(* IEC 61131-3 sources: simple-control-modules/src/Bulbs, 3 files *)

(* ---- Colors.st ---- *)
NAMESPACE Simatic.Ax.SimpleControlModules
    TYPE
        Colors : (Red, Green, Blue, Yellow);
    END_TYPE

END_NAMESPACE

(* ---- Bulb.st ---- *)
USING Simatic.Ax.Io.Output;
USING Simatic.Ax.Io.Input;

NAMESPACE Simatic.Ax.SimpleControlModules

    /// Class to handle a bulb
    CLASS Bulb
        VAR PUBLIC
            Output : ItfBinOutput;
        END_VAR

        /// Switch the lamp on (value := TRUE) or off (value := FALSE)
        /// value : Value to set
        METHOD PUBLIC Set
            VAR_INPUT
                value : bool;
            END_VAR
            IF (Output = NULL) THEN
                RETURN;
            END_IF;
            Output.SetQ(value := value);

        END_METHOD

        /// Switch the lamp on
        METHOD PUBLIC SwitchOn
            IF (Output = NULL) THEN
                RETURN;
            END_IF;
            Output.SetQ(value := TRUE);
        END_METHOD

        /// Switch the lamp off
        METHOD PUBLIC SwitchOff
            IF (Output = NULL) THEN
                RETURN;
            END_IF;
            Output.SetQ(value := FALSE);
        END_METHOD

        /// Toggle the lamp
        METHOD PUBLIC Toggle
            IF (Output = NULL) THEN
                RETURN;
            END_IF;
            Output.Toggle();
        END_METHOD

    END_CLASS
END_NAMESPACE

(* ---- LightStack.st ---- *)
USING Simatic.Ax.IO.Output;

NAMESPACE Simatic.Ax.SimpleControlModules

    /// Class of a lightstack with 3 lamps (Red, Yellow, Green)

    CLASS LightStackRdYeGnBl
        VAR PUBLIC
            QRed : ItfBinOutput;
            QYellow : ItfBinOutput;
            QGreen : ItfBinOutput;
            QBlue : ItfBinOutput;
        END_VAR

        /// Switch on the lamp of color c

        METHOD PUBLIC SwitchOn
            VAR_INPUT
                c : Colors;
            END_VAR;
            CASE c OF
                Colors#Red      : QRed.SetOn();
                Colors#Yellow   : QYellow.SetOn();
                Colors#Green    : QGreen.SetOn();
                Colors#Blue     : QBlue.SetOn();
            ELSE
                ;
            END_CASE;

        END_METHOD

        /// Switch off the lamp of color c

        METHOD PUBLIC SwitchOff
            VAR_INPUT
                c : Colors;
            END_VAR;
            CASE c OF
                Colors#Red      : QRed.SetOff();
                Colors#Yellow   : QYellow.SetOff();
                Colors#Green    : QGreen.SetOff();
                Colors#Blue     : QBlue.SetOff();
            ELSE
                ;
            END_CASE;

        END_METHOD

        METHOD PUBLIC GetState : BOOL
            VAR_INPUT
                c : Colors;
            END_VAR
            VAR_TEMP
                q : BOOL;
            END_VAR
            CASE c OF
                Colors#Red      : GetState := QRed.IsOn();
                Colors#Yellow   : GetState := QYellow.IsOn();
                Colors#Green    : GetState := QGreen.IsOn();
                Colors#Blue     : GetState := QBlue.IsOn();
            ELSE
                GetState := FALSE;
            END_CASE;

        END_METHOD

    END_CLASS
END_NAMESPACE
